# EPICS substitutions: examplesTop/ndsex1App/Db/DevicePVs.substitutions
file "nds3_DevicePV.template" {
pattern
{
    BOARDTYPE,
    BOARDTYPEIDX,
    CBS1,
    CBS2,
    DEVICEPV_NAME,
}

{
    "B",
    "0",
    "TEST",
    "FCT0",
    "DevicePVs",
}

}
